Yaskawa INFORM job: OK_R2_O55B(90,0)KMOK_HARDOX.JBI

/JOB
//NAME OK_R2_O55B(90,0)KMOK_HARDOX
//POS
///NPOS 288,288,288,21,0,0
///TOOL 0
///POSTYPE PULSE
///PULSE
C00000=-9957,-80120,-66349,29251,62843,-41580
C00001=-119270,-98989,-86741,-6328,68520,-73858
C00002=-119780,-37820,-56111,-5839,80997,-74654
C00003=-120049,20077,-10457,-5740,82625,-74818
C00004=-144319,37014,-5855,2257,77898,-81650
C00005=-140529,51042,7974,-9565,85073,-64090
C00006=-140529,50609,8792,-9570,84355,-64035
C00007=-140529,50663,8686,-9570,84448,-64042
C00008=-140735,53191,11473,-9511,84012,-64075
C00009=-140529,50663,8686,-9570,84448,-64042
C00010=-132608,43274,6223,-26925,79302,-63189
C00011=-133562,42203,5091,-26579,79144,-63498
C00012=-132608,43724,5035,-26857,80165,-63389
C00013=-141550,80814,37938,-2920,95813,-64462
C00014=-141396,81120,39088,-2939,95269,-64399
C00015=-141396,80823,39851,-2936,94645,-64387
C00016=-141396,80877,39711,-2936,94757,-64389
C00017=-141226,78223,36470,-2964,95394,-64348
C00018=-141396,80877,39711,-2936,94757,-64389
C00019=-140829,81512,40491,-3016,94624,-64202
C00020=-140134,82102,41214,-3116,94504,-63971
C00021=-140829,81912,39485,-3022,95448,-64222
C00022=-137405,-31621,-64154,-15278,80257,-65243
C00023=-140140,-48602,-70983,-11254,71048,-74410
C00024=-141076,-49933,-70540,-10875,69988,-74633
C00025=-141076,-50277,-69406,-10930,69130,-74550
C00026=-141076,-50226,-69587,-10919,69267,-74563
C00027=-141467,-47373,-67920,-10702,69651,-74733
C00028=-141076,-50226,-69587,-10919,69267,-74563
C00029=-141874,-50689,-69854,-10542,69093,-74827
C00030=-143117,-51074,-70075,-9948,68881,-75243
C00031=-141874,-50354,-70946,-10488,69924,-74901
C00032=-147268,-6347,-50211,3630,100062,-76353
C00033=-146938,-6418,-49322,3551,99466,-76267
C00034=-146938,-6964,-48693,3545,98802,-76289
C00035=-146938,-6869,-48804,3545,98917,-76285
C00036=-146728,-9231,-50671,3485,98843,-76222
C00037=-146938,-6869,-48804,3545,98917,-76285
C00038=-151923,-27684,-59821,11781,84663,-77431
C00039=-150653,-27440,-59655,11346,84518,-77042
C00040=-151923,-26904,-61083,11768,85817,-77322
C00041=-127144,-21020,-54073,-16205,79799,-73423
C00042=-126838,-21905,-54390,-16337,79609,-73295
C00043=-126838,-22307,-53617,-16368,78953,-73207
C00044=-126838,-22196,-53838,-16359,79138,-73232
C00045=-124787,-22488,-54046,-17172,79509,-72603
C00046=-124787,-22654,-53716,-17186,79233,-72564
C00047=-125689,-22541,-53635,-16830,79066,-72840
C00048=-125495,-21030,-56345,-16804,81448,-73105
C00049=-137099,-135087,-110065,-14474,54639,-73776
C00050=-134884,-135911,-107803,-15875,53297,-72629
C00051=-134884,-134891,-106174,-15972,52835,-72554
C00052=-134884,-135228,-106712,-15940,52987,-72578
C00053=-129865,-136478,-107050,-18378,53628,-70507
C00054=-129865,-135962,-106251,-18430,53413,-70467
C00055=-131869,-135536,-106136,-17475,53114,-71287
C00056=-131377,-137376,-108864,-17542,53921,-71215
C00057=-139724,-149069,-111841,-14344,48265,-73992
C00058=-138735,-146286,-108991,-14933,48130,-73516
C00059=-138325,-143626,-108337,-14931,49139,-73488
C00060=-138410,-146030,-110862,-14819,49432,-73572
C00061=-176899,-100061,-98449,5916,63407,-89727
C00062=-179900,-97566,-95391,7380,63058,-90869
C00063=-179900,-97456,-94205,7424,62390,-90913
C00064=-179900,-97485,-94494,7413,62551,-90902
C00065=-169343,-119267,-96895,-8817,44711,-86747
C00066=-169343,-119018,-96376,-8846,44521,-86728
C00067=-168683,-117584,-95925,-9230,45055,-86464
C00068=-169216,-119583,-98076,-8807,45288,-86741
C00069=-162548,-60984,-74877,-11016,61707,-85538
C00070=-184352,-15408,-50569,-7993,71565,-76848
C00071=-184633,-15854,-49265,-7894,70519,-76872
C00072=-184633,-16240,-48510,-7925,69861,-76830
C00073=-184633,-16157,-48676,-7919,70004,-76840
C00074=-184233,-13625,-46764,-8123,70163,-76718
C00075=-184633,-16157,-48676,-7919,70004,-76840
C00076=-187381,11831,-34077,-2210,90888,-77611
C00077=-186375,11183,-34661,-2532,90938,-77309
C00078=-187381,12466,-34757,-2212,91632,-77624
C00079=-182192,42266,-7795,-19168,104635,-71349
C00080=-189067,53591,3425,-6745,109963,-71903
C00081=-189067,53103,3970,-6717,109382,-71871
C00082=-189067,53201,3857,-6722,109501,-71876
C00083=-189450,50860,1262,-6719,109865,-72023
C00084=-189067,53201,3857,-6722,109501,-71876
C00085=-185034,14321,-30270,-13993,89133,-70711
C00086=-186120,15304,-29370,-13637,88918,-71028
C00087=-185035,15000,-31072,-14012,89952,-70804
C00088=-182682,60735,12692,-23773,101105,-73169
C00089=-182682,60735,12692,-23773,101105,-73169
C00090=-183650,63040,17037,-21830,101290,-73190
C00091=-183650,62538,17836,-21764,100591,-73060
C00092=-183650,62598,17737,-21771,100675,-73076
C00093=-183528,62176,17250,-21794,100781,-73054
C00094=-183650,63460,16427,-21883,101838,-73293
C00095=-189227,48884,3,-21319,102940,-75405
C00096=-189468,47971,159,-21225,102357,-75379
C00097=-189468,47380,928,-21153,101633,-75249
C00098=-189468,47470,808,-21165,101744,-75269
C00099=-189367,47114,422,-21186,101818,-75248
C00100=-189432,48469,-714,-21310,103107,-75504
C00101=-175013,33301,-13153,-29999,98235,-49044
C00102=-175115,31766,-13036,-29901,97452,-48874
C00103=-175115,31283,-12339,-29848,96864,-48718
C00104=-175115,31366,-12461,-29858,96964,-48746
C00105=-176020,31704,-12122,-29658,96640,-48987
C00106=-175115,31366,-12461,-29858,96964,-48746
C00107=-177389,49548,3663,-27032,106629,-51330
C00108=-177525,47289,1207,-27077,106904,-51447
C00109=-177389,50188,2794,-27172,107402,-51519
C00110=-188015,41028,-12957,-12549,102183,-51760
C00111=-188146,40613,-11827,-12473,101279,-51708
C00112=-188165,40048,-11193,-12432,100612,-51645
C00113=-188165,40130,-11271,-12438,100700,-51655
C00114=-187344,39553,-11878,-12615,100887,-51416
C00115=-188165,40130,-11271,-12438,100700,-51655
C00116=-187875,42015,-9279,-12487,100489,-51542
C00117=-187566,44182,-6969,-12539,100230,-51416
C00118=-187875,42842,-10030,-12532,101356,-51631
C00119=-171459,-4614,-45398,-33605,84930,-48191
C00120=-170900,-6042,-43653,-33882,83616,-47589
C00121=-170900,-6530,-42846,-33920,82989,-47396
C00122=-170900,-6366,-43125,-33907,83204,-47461
C00123=-169534,-6797,-43470,-34394,83698,-47104
C00124=-169534,-7027,-43077,-34411,83398,-47011
C00125=-170096,-6658,-42784,-34212,83197,-47160
C00126=-169785,-6714,-43972,-34288,83898,-47260
C00127=-170398,9353,-32178,-34027,84507,-47673
C00128=-170215,8790,-30856,-34141,83656,-47346
C00129=-170215,8459,-30301,-34168,83233,-47218
C00130=-170215,8580,-30507,-34158,83391,-47266
C00131=-168835,8055,-30970,-34644,83914,-46912
C00132=-168835,7853,-30623,-34659,83653,-46831
C00133=-169290,8275,-30251,-34499,83472,-46947
C00134=-169213,8760,-31391,-34484,84292,-47173
C00135=-186069,25736,-27642,1526,92687,-58921
C00136=-186694,24000,-25961,1734,90774,-59129
C00137=-186694,23425,-25397,1733,90131,-59136
C00138=-186694,23662,-25633,1733,90398,-59133
C00139=-187283,19938,-29188,1932,90686,-59306
C00140=-187283,19583,-28837,1932,90288,-59311
C00141=-187018,21055,-27442,1842,90183,-59234
C00142=-187095,21607,-28285,1869,90987,-59245
C00143=-183298,20097,-29492,20792,92835,-75129
C00144=-182431,19002,-28896,20491,91770,-75035
C00145=-182431,18218,-28039,20473,90895,-75182
C00146=-182431,18445,-28295,20478,91152,-75138
C00147=-182795,15268,-31245,20599,91404,-75212
C00148=-182795,14938,-30873,20592,91029,-75276
C00149=-182620,16002,-29895,20535,90939,-75235
C00150=-182918,16284,-31560,20654,92104,-75132
C00151=-186265,48055,-1212,11796,87124,-79966
C00152=-186965,48573,-100,12039,86806,-80215
C00153=-186965,47910,713,12044,85983,-80295
C00154=-186965,47988,613,12044,86082,-80285
C00155=-186694,50137,2964,11952,85709,-80238
C00156=-186965,47988,613,12044,86082,-80285
C00157=-183974,61337,12156,5178,92575,-80151
C00158=-184645,62112,13036,5353,92472,-80362
C00159=-183974,61852,11573,5182,93194,-80123
C00160=-179887,91143,39097,3384,105716,-79096
C00161=-179840,89635,38790,3370,105129,-79098
C00162=-179840,89143,39323,3359,104550,-79112
C00163=-179840,89220,39235,3359,104642,-79110
C00164=-180024,86327,35591,3386,105404,-79148
C00165=-179840,89220,39235,3359,104642,-79110
C00166=-186520,62301,10800,17886,95759,-79423
C00167=-185837,61712,10122,17722,95736,-79206
C00168=-186520,62996,10143,17919,96484,-79317
C00169=-174567,29627,-16130,-6089,77714,-79974
C00170=-174267,31304,-12949,-6249,76643,-79825
C00171=-179026,33960,-10363,-4044,76139,-81308
C00172=-179026,33960,-10363,-4044,76139,-81308
C00173=-174024,52452,5562,-15282,87335,-82643
C00174=-181124,73254,24397,-458,98517,-83064
C00175=-182896,88636,42871,4243,102910,-77228
C00176=-180140,85434,39000,4081,103513,-76295
C00177=-180140,85434,39000,4081,103513,-76295
C00178=-184647,66871,19208,14888,96534,-76534
C00179=-174267,31304,-12949,-6249,76643,-79825
C00180=-174494,31610,-14990,-6114,78032,-79964
C00181=-175013,33301,-13153,-29999,98235,-49044
C00182=-175343,30235,-14768,-29874,97621,-48999
C00183=-171906,8512,-28233,-36021,84269,-45281
C00184=-172758,8115,-27337,-35775,83319,-45298
C00185=-172255,16606,-19687,-35958,83238,-45074
C00186=-171987,21177,-15407,-36061,83112,-44927
C00187=-171987,21177,-15407,-36061,83112,-44927
C00188=-180391,49402,2354,-18177,99354,-48334
C00189=-181669,75195,30349,-14733,108937,-58802
C00190=-184056,79778,35948,-11160,112261,-59402
C00191=-184907,70087,24268,-11430,114320,-59912
C00192=-184907,70087,24268,-11430,114320,-59912
C00193=-179652,49581,2539,-22463,107252,-59131
C00194=-172758,8115,-27337,-35775,83319,-45298
C00195=-172634,8341,-28512,-35775,84058,-45486
C00196=-153759,-18914,-52407,-41335,92413,-41016
C00197=-152540,-20147,-51692,-41605,92133,-40401
C00198=-152993,-17865,-48148,-41450,91166,-40203
C00199=-159302,-18488,-48629,-39831,88393,-41734
C00200=-159302,-18488,-48629,-39831,88393,-41734
C00201=-166414,13220,-30767,-32137,108347,-48872
C00202=-176872,12138,-36686,-11233,108343,-73701
C00203=-180381,23244,-27161,-3143,115050,-73458
C00204=-177105,21284,-28961,-3234,115264,-72371
C00205=-177105,21284,-28961,-3234,115264,-72371
C00206=-175157,7036,-41533,-6172,108047,-57119
C00207=-152993,-17864,-48148,-41450,91166,-40203
C00208=-153162,-17915,-50375,-41466,92114,-40650
C00209=-157956,-50140,-75109,2057,72313,-66630
C00210=-160224,-49369,-73518,3152,71800,-67393
C00211=-160503,-46712,-70493,3295,71314,-67502
C00212=-152523,-45623,-69844,-552,71345,-64837
C00213=-152523,-45623,-69844,-552,71345,-64837
C00214=-148927,-14811,-56631,-4403,95378,-64978
C00215=-148763,-1156,-47820,-3788,104699,-80082
C00216=-148630,8941,-39588,-6498,110680,-80853
C00217=-152650,7748,-40640,-6101,110438,-82132
C00218=-152650,7748,-40640,-6101,110438,-82132
C00219=-155137,-28863,-64381,-3266,86260,-82126
C00220=-160503,-46712,-70493,3295,71314,-67502
C00221=-160802,-46385,-74012,3397,73655,-67536
C00222=-183650,63040,17037,-21830,101290,-73190
C00223=-181574,69704,24792,-21980,100549,-72331
C00224=-183403,72450,28416,-19365,101992,-72790
C00225=-183309,72093,27990,-19380,102088,-72773
C00226=-183520,72890,28942,-19345,101875,-72811
C00227=-183958,70615,26232,-19347,102249,-73025
C00228=-183958,70934,25678,-19391,102726,-73103
C00229=-192384,50426,1269,-3472,96407,-72620
C00230=-192384,50016,1751,-3467,95901,-72606
C00231=-184117,69898,25781,-20658,102920,-73473
C00232=-190944,51922,5194,-20323,104561,-76131
C00233=-191415,50867,4029,-20288,104619,-76303
C00234=-193520,46467,-770,-20112,104798,-77054
C00235=-193520,47017,-1447,-20188,105457,-77168
C00236=-171741,3085,-44079,-22866,113958,-71236
C00237=-130348,29463,-19685,-22297,122832,-57661
C00238=-129735,-75595,-89571,-13565,72601,-49374
C00239=-143928,-62129,-81754,5565,77375,-52115
C00240=-142081,-63272,-82268,4854,76992,-51525
C00241=-142081,-63272,-82268,4854,76992,-51525
C00242=-127755,-87223,-86704,-10460,53798,-73673
C00243=-115599,-84167,-82164,-28839,54869,-69627
C00244=-115830,-77465,-79174,-28196,56209,-70126
C00245=-120569,18950,-14128,-20651,63759,-73413
C00246=-120570,21073,-12131,-20673,63629,-73389
C00247=-120570,21641,-13746,-20463,64836,-73615
C00248=-131610,1281,-36986,-13629,66366,-77786
C00249=-142543,23012,-23162,1458,80523,-80349
C00250=-139525,20137,-20065,-7610,74683,-81021
C00251=-142876,20525,-19823,1343,74165,-80532
C00252=-139662,22596,-17854,-198,73998,-79499
C00253=-139662,22596,-17854,-198,73998,-79499
C00254=-141793,37019,-7971,5655,84578,-79297
C00255=-137277,64767,17706,-3970,99490,-79285
C00256=-134924,69316,23645,-11495,101419,-79759
C00257=-137432,66658,20404,-11237,101707,-80615
C00258=-137432,66658,20404,-11237,101707,-80615
C00259=-140896,36331,-9506,-5892,87094,-79888
C00260=-139525,20137,-20065,-7610,74683,-81021
C00261=-139348,19632,-23053,-7644,76265,-81063
C00262=-132254,-67818,-87549,-11183,71854,-78389
C00263=-159615,-10281,-58898,-7636,100535,-90235
C00264=-166998,7770,-33829,-38669,93984,-50545
C00265=-168265,5123,-34621,-38271,92780,-50607
C00266=-168071,5758,-34073,-38323,92849,-50556
C00267=-167928,7434,-32586,-38359,92864,-50506
C00268=-172719,9530,-31332,-27823,83706,-47451
C00269=-172719,9530,-31332,-27823,83706,-47451
C00270=-172320,11286,-29764,-27974,83774,-47329
C00271=-179459,29271,-20356,-13837,95701,-48796
C00272=-183465,26284,-23592,-4892,94989,-48302
C00273=-181920,25197,-24652,-5328,95168,-47844
C00274=-174479,31677,-20338,1503,103987,-43795
C00275=-180212,26004,-22183,17305,100653,-42977
C00276=-181024,26764,-23793,17575,102127,-43022
C00277=-174949,-10425,-55605,-83,88665,-45823
C00278=-166426,-64689,-90076,-3246,82158,-43137
C00279=-131468,-82914,-92239,-33517,76500,-33632
C00280=-132751,-79712,-87299,-33282,74833,-33639
C00281=-135289,-78928,-86943,-32417,74029,-34418
C00282=-167985,-50339,-72512,-17957,69595,-45682
C00283=-161662,-56646,-68227,-34204,59627,-42917
C00284=-161369,-58109,-70614,-34130,60339,-43034
C00285=-153489,-114383,-104764,-40748,57378,-38072
C00286=-152369,-109512,-103102,-40646,59036,-38246
C00287=-7483,-109512,-100434,-40646,59036,-38246
BC00000=15,674025,1075175
BC00001=140466,674228,172767
BC00002=140466,729284,172767
BC00003=140466,791751,172767
BC00004=182866,791751,67340
BC00005=182866,791751,67340
BC00006=182866,791751,67340
BC00007=182866,791751,67340
BC00008=182866,791751,67340
BC00009=182866,791751,67340
BC00010=182866,791751,67340
BC00011=182866,791751,67340
BC00012=182866,791751,67340
BC00013=182866,791751,67340
BC00014=182866,791751,67340
BC00015=182866,791751,67340
BC00016=182866,791751,67340
BC00017=182866,791751,67340
BC00018=182866,791751,67340
BC00019=182866,791751,67340
BC00020=182866,791751,67340
BC00021=182866,791751,67340
BC00022=182866,791752,67339
BC00023=182866,791752,67339
BC00024=182866,791752,67339
BC00025=182866,791752,67339
BC00026=182866,791752,67339
BC00027=182866,791752,67339
BC00028=182866,791752,67339
BC00029=182866,791752,67339
BC00030=182866,791752,67339
BC00031=182866,791752,67339
BC00032=182866,791752,67339
BC00033=182866,791752,67339
BC00034=182866,791752,67339
BC00035=182866,791752,67339
BC00036=182866,791752,67337
BC00037=182866,791752,67339
BC00038=182866,791752,67339
BC00039=182866,791752,67339
BC00040=182866,791752,67339
BC00041=182866,791752,67339
BC00042=182866,791752,67339
BC00043=182866,791752,67339
BC00044=182866,791752,67339
BC00045=182866,791752,67339
BC00046=182866,791752,67339
BC00047=182866,791752,67339
BC00048=182866,791752,67339
BC00049=182866,791752,67339
BC00050=182866,791752,67339
BC00051=182866,791752,67339
BC00052=182866,791752,67339
BC00053=182866,791752,67339
BC00054=182866,791752,67339
BC00055=182866,791752,67339
BC00056=182866,791752,67339
BC00057=182866,791752,67339
BC00058=182866,791752,67339
BC00059=182866,791752,67339
BC00060=182866,791752,67339
BC00061=182866,791752,67339
BC00062=182866,791752,67339
BC00063=182866,791752,67339
BC00064=182866,791752,67339
BC00065=182866,791752,67339
BC00066=182866,791752,67339
BC00067=182865,791751,67336
BC00068=182865,791751,67336
BC00069=182865,791751,67336
BC00070=248959,799596,47476
BC00071=248959,799596,47476
BC00072=248959,799596,47476
BC00073=248959,799596,47476
BC00074=248959,799596,47476
BC00075=248959,799596,47476
BC00076=248959,799596,47476
BC00077=248959,799596,47476
BC00078=248959,799596,47476
BC00079=248959,799596,47476
BC00080=248959,799596,47476
BC00081=248959,799596,47476
BC00082=248959,799596,47476
BC00083=248959,799596,47476
BC00084=248959,799596,47476
BC00085=248959,799596,47476
BC00086=248959,799596,47476
BC00087=248959,799596,47475
BC00088=248959,799596,47475
BC00089=248959,799596,47475
BC00090=248959,799596,47475
BC00091=248959,799596,47475
BC00092=248959,799596,47475
BC00093=248959,799596,47475
BC00094=248959,799596,47475
BC00095=248959,799596,47475
BC00096=248959,799596,47475
BC00097=248959,799596,47475
BC00098=248959,799596,47475
BC00099=248959,799596,47475
BC00100=248959,799596,47475
BC00101=203274,799596,47475
BC00102=203274,799596,47475
BC00103=203274,799596,47475
BC00104=203274,799596,47475
BC00105=203274,799596,47475
BC00106=203274,799596,47475
BC00107=203274,799596,47475
BC00108=203274,799596,47475
BC00109=203274,799596,47475
BC00110=209362,813826,28785
BC00111=209362,813826,28785
BC00112=209362,813826,28785
BC00113=209362,813826,28785
BC00114=209362,813826,28785
BC00115=209362,813826,28785
BC00116=209362,813826,28785
BC00117=209362,813826,28784
BC00118=209362,813826,28785
BC00119=209362,813826,28785
BC00120=209362,813826,28785
BC00121=209362,813826,28785
BC00122=209362,813826,28785
BC00123=209362,813826,28785
BC00124=209362,813826,28785
BC00125=209362,813826,28785
BC00126=209362,813826,28785
BC00127=209362,813826,28785
BC00128=209362,813826,28785
BC00129=209362,813826,28785
BC00130=209362,813826,28785
BC00131=209362,813826,28785
BC00132=209362,813826,28785
BC00133=209362,813826,28785
BC00134=209362,813826,28785
BC00135=209362,813826,28784
BC00136=209362,813826,28784
BC00137=209362,813826,28784
BC00138=209362,813826,28784
BC00139=209362,813826,28784
BC00140=209362,813826,28784
BC00141=209362,813826,28784
BC00142=209362,813826,28784
BC00143=209362,813826,28784
BC00144=209362,813826,28784
BC00145=209362,813826,28784
BC00146=209362,813826,28784
BC00147=209362,813826,28784
BC00148=209362,813826,28784
BC00149=209362,813826,28784
BC00150=209362,813826,28784
BC00151=209363,813827,28780
BC00152=209363,813827,28780
BC00153=209363,813827,28780
BC00154=209363,813827,28780
BC00155=209363,813827,28780
BC00156=209363,813827,28780
BC00157=209363,813827,28780
BC00158=209363,813827,28780
BC00159=209363,813827,28780
BC00160=209363,813827,1884
BC00161=209363,813827,1884
BC00162=209363,813827,1884
BC00163=209363,813827,1884
BC00164=209363,813827,1884
BC00165=209363,813827,1884
BC00166=209363,813827,1884
BC00167=209363,813827,1884
BC00168=209363,813827,1884
BC00169=209363,813827,28780
BC00170=209363,813827,28780
BC00171=209363,813827,28780
BC00172=209363,813827,28780
BC00173=209363,813827,28780
BC00174=209363,813827,28780
BC00175=209363,813827,28776
BC00176=209363,813827,28776
BC00177=209363,813827,28776
BC00178=209363,813827,28776
BC00179=209363,813827,28780
BC00180=209363,813827,28780
BC00181=203274,799596,47475
BC00182=203274,799596,47475
BC00183=203274,799596,47475
BC00184=203274,799596,47475
BC00185=203274,799596,47475
BC00186=203275,799597,47472
BC00187=203275,799597,47472
BC00188=203275,799597,47472
BC00189=203275,799597,47471
BC00190=203275,799597,47471
BC00191=203275,799597,47470
BC00192=203275,799597,47470
BC00193=203275,799597,47470
BC00194=203274,799596,47475
BC00195=203275,799596,47475
BC00196=203275,799596,47475
BC00197=203275,799596,47474
BC00198=203275,799596,47474
BC00199=203275,799596,47474
BC00200=203275,799596,47474
BC00201=203275,799596,47474
BC00202=203275,799596,47474
BC00203=203275,799596,47474
BC00204=203275,799596,47474
BC00205=203275,799596,47474
BC00206=203275,799596,47474
BC00207=203275,799596,47474
BC00208=203275,799596,47474
BC00209=203275,799596,47474
BC00210=203275,799596,47474
BC00211=203275,799596,47474
BC00212=203275,799596,47474
BC00213=203275,799596,47474
BC00214=203275,799596,47474
BC00215=203275,799596,47474
BC00216=203275,799596,47474
BC00217=203275,799596,47474
BC00218=203275,799596,47474
BC00219=203275,799596,47474
BC00220=203275,799596,47474
BC00221=203275,799596,47474
BC00222=248959,799596,47475
BC00223=248959,799596,47475
BC00224=248959,799596,47475
BC00225=248959,799596,47475
BC00226=248959,799596,47475
BC00227=248959,799596,47475
BC00228=248959,799596,47475
BC00229=248959,799596,47475
BC00230=248959,799596,47475
BC00231=248959,799596,47475
BC00232=248959,799596,47475
BC00233=248959,799596,47475
BC00234=248959,799596,47475
BC00235=248959,799596,47475
BC00236=248959,799596,47475
BC00237=169428,732562,47475
BC00238=169431,732564,47474
BC00239=169431,732564,47474
BC00240=169431,732564,47474
BC00241=169431,732564,47474
BC00242=169431,732564,47474
BC00243=169431,732564,47474
BC00244=169431,732564,47474
BC00245=172916,732564,47474
BC00246=172916,732564,47474
BC00247=172916,732564,47474
BC00248=172916,804432,47474
BC00249=172916,804432,47474
BC00250=172916,804432,47473
BC00251=172916,804432,47473
BC00252=172916,804432,47473
BC00253=172916,804432,47473
BC00254=172916,804432,47473
BC00255=172916,804432,47473
BC00256=172916,804432,47473
BC00257=172916,804432,47473
BC00258=172916,804432,47473
BC00259=172916,804432,47473
BC00260=172916,804432,47473
BC00261=172916,804432,47473
BC00262=172916,804432,47473
BC00263=172916,804432,47473
BC00264=209362,813826,28785
BC00265=209362,813826,28785
BC00266=209362,813826,28785
BC00267=209362,813826,28785
BC00268=209362,813826,28785
BC00269=209362,813826,28785
BC00270=209362,813826,28785
BC00271=209362,813826,28785
BC00272=209362,813826,28785
BC00273=209362,813826,28785
BC00274=209362,813826,28785
BC00275=209362,813826,28785
BC00276=209362,813826,28785
BC00277=209362,813826,28785
BC00278=209362,813826,28785
BC00279=209362,755898,28785
BC00280=209362,755898,28785
BC00281=209362,755898,28785
BC00282=209362,755898,28785
BC00283=209362,755898,28785
BC00284=209362,755898,28785
BC00285=209362,755898,28785
BC00286=209362,675971,28785
BC00287=209362,663746,462190
EC00000=798156,0
EC00001=798153,2
EC00002=798153,2
EC00003=798153,2
EC00004=798153,2
EC00005=798153,2
EC00006=798153,2
EC00007=798153,2
EC00008=798153,2
EC00009=798153,2
EC00010=798153,2
EC00011=798153,2
EC00012=798153,2
EC00013=798153,2
EC00014=798153,2
EC00015=798153,2
EC00016=798153,2
EC00017=798153,2
EC00018=798153,2
EC00019=798153,2
EC00020=798153,2
EC00021=798153,2
EC00022=798152,3
EC00023=798152,3
EC00024=798152,3
EC00025=798152,3
EC00026=798152,3
EC00027=798152,3
EC00028=798152,3
EC00029=798152,3
EC00030=798152,3
EC00031=798152,3
EC00032=798152,3
EC00033=798152,3
EC00034=798152,3
EC00035=798152,3
EC00036=798151,3
EC00037=798152,3
EC00038=798152,3
EC00039=798152,3
EC00040=798152,3
EC00041=798152,3
EC00042=798152,3
EC00043=798152,3
EC00044=798152,3
EC00045=798152,3
EC00046=798152,3
EC00047=798152,3
EC00048=798152,3
EC00049=798152,3
EC00050=798152,3
EC00051=798152,3
EC00052=798152,3
EC00053=798152,3
EC00054=798152,3
EC00055=798152,3
EC00056=798152,3
EC00057=798152,3
EC00058=798152,3
EC00059=798152,3
EC00060=798152,3
EC00061=798152,3
EC00062=798152,3
EC00063=798152,3
EC00064=798152,3
EC00065=798152,3
EC00066=798152,3
EC00067=798151,3
EC00068=798151,3
EC00069=798151,3
EC00070=798151,3
EC00071=798151,3
EC00072=798151,3
EC00073=798151,3
EC00074=798151,3
EC00075=798151,3
EC00076=798151,3
EC00077=798151,3
EC00078=798151,3
EC00079=798151,3
EC00080=798151,3
EC00081=798151,3
EC00082=798151,3
EC00083=798151,3
EC00084=798151,3
EC00085=798151,3
EC00086=798151,3
EC00087=798150,4
EC00088=798150,4
EC00089=798150,4
EC00090=798150,4
EC00091=798150,4
EC00092=798150,4
EC00093=798150,4
EC00094=798150,4
EC00095=798150,4
EC00096=798150,4
EC00097=798149,4
EC00098=798149,4
EC00099=798149,4
EC00100=798149,4
EC00101=798148,4
EC00102=798148,4
EC00103=798148,4
EC00104=798148,4
EC00105=798148,4
EC00106=798148,4
EC00107=798148,4
EC00108=798148,4
EC00109=798148,4
EC00110=798148,4
EC00111=798148,4
EC00112=798148,4
EC00113=798148,4
EC00114=798148,4
EC00115=798148,4
EC00116=798148,4
EC00117=798147,5
EC00118=798148,4
EC00119=798148,4
EC00120=798148,4
EC00121=798148,4
EC00122=798148,4
EC00123=798148,4
EC00124=798148,4
EC00125=798148,4
EC00126=798148,4
EC00127=798148,4
EC00128=798148,4
EC00129=798148,4
EC00130=798148,4
EC00131=798148,4
EC00132=798148,4
EC00133=798148,4
EC00134=798148,4
EC00135=798147,4
EC00136=798147,4
EC00137=798147,4
EC00138=798147,4
EC00139=798147,4
EC00140=798147,4
EC00141=798147,4
EC00142=798147,4
EC00143=798147,4
EC00144=798147,4
EC00145=798147,4
EC00146=798147,4
EC00147=798147,4
EC00148=798147,4
EC00149=798147,4
EC00150=798147,4
EC00151=798145,8
EC00152=798145,8
EC00153=798145,8
EC00154=798145,8
EC00155=798145,8
EC00156=798145,8
EC00157=798145,8
EC00158=798145,8
EC00159=798145,8
EC00160=798145,8
EC00161=798145,8
EC00162=798145,8
EC00163=798145,8
EC00164=798145,8
EC00165=798145,8
EC00166=798145,8
EC00167=798145,8
EC00168=798145,8
EC00169=798145,8
EC00170=798145,8
EC00171=798145,11
EC00172=798145,11
EC00173=798145,11
EC00174=798145,11
EC00175=798144,11
EC00176=798144,11
EC00177=798144,11
EC00178=798144,11
EC00179=798145,8
EC00180=798145,8
EC00181=798148,4
EC00182=798148,4
EC00183=798148,4
EC00184=798148,4
EC00185=798148,4
EC00186=798147,4
EC00187=798147,4
EC00188=798147,4
EC00189=798145,5
EC00190=798145,5
EC00191=798144,6
EC00192=798144,6
EC00193=798144,6
EC00194=798148,4
EC00195=798147,4
EC00196=798147,4
EC00197=798146,5
EC00198=798146,5
EC00199=798146,5
EC00200=798146,5
EC00201=798146,5
EC00202=798146,5
EC00203=798146,5
EC00204=798146,5
EC00205=798146,5
EC00206=798146,5
EC00207=798146,5
EC00208=798146,5
EC00209=798146,5
EC00210=798146,5
EC00211=798146,5
EC00212=798146,5
EC00213=798146,5
EC00214=798146,5
EC00215=798146,5
EC00216=798146,5
EC00217=798146,5
EC00218=798146,5
EC00219=798146,5
EC00220=798146,5
EC00221=798146,5
EC00222=798150,4
EC00223=798150,4
EC00224=798150,4
EC00225=798150,4
EC00226=798150,4
EC00227=798150,4
EC00228=798150,4
EC00229=798150,4
EC00230=798150,4
EC00231=798150,4
EC00232=798150,4
EC00233=798150,4
EC00234=798150,4
EC00235=798150,4
EC00236=798150,4
EC00237=798150,4
EC00238=798148,13
EC00239=798148,13
EC00240=798148,13
EC00241=798148,13
EC00242=798148,13
EC00243=798148,13
EC00244=798148,13
EC00245=798148,13
EC00246=798148,13
EC00247=798148,13
EC00248=798148,13
EC00249=798148,13
EC00250=798147,13
EC00251=798147,13
EC00252=798147,13
EC00253=798147,13
EC00254=798147,13
EC00255=798147,13
EC00256=798147,13
EC00257=798147,13
EC00258=798147,13
EC00259=798147,13
EC00260=798147,13
EC00261=798147,13
EC00262=798147,13
EC00263=798147,13
EC00264=798148,4
EC00265=798148,4
EC00266=798148,4
EC00267=798148,4
EC00268=798148,4
EC00269=798148,4
EC00270=798148,4
EC00271=798148,4
EC00272=798148,4
EC00273=798148,4
EC00274=798148,4
EC00275=798148,4
EC00276=798148,4
EC00277=798148,4
EC00278=798148,4
EC00279=798148,4
EC00280=798148,4
EC00281=798148,4
EC00282=798148,4
EC00283=798148,4
EC00284=798148,4
EC00285=798148,4
EC00286=798148,4
EC00287=798148,4
///POSTYPE BASE
///RECTAN
///RCONF 0,0,0,0,0,0,0,0,0,0,0,0,0,0,0,0,0,0,0,0,0,0,0,0
P00006=0.222,-3.123,-1.508,0.0000,0.0000,0.0000
P00021=-0.225,-6.128,-0.405,0.0000,0.0000,0.0000
P00022=0.222,-3.123,-1.508,0.0000,0.0000,0.0000
P00023=0.143,-0.036,0.682,0.0000,0.0000,0.0000
P00024=0.145,-0.552,1.326,0.0000,0.0000,0.0000
P00025=-2.003,0.006,0.728,0.0000,0.0000,0.0000
P00026=0.562,-0.002,-0.337,0.0000,0.0000,0.0000
P00027=-0.746,0.015,-9.096,0.0000,0.0000,0.0000
P00028=-2.237,-0.018,-7.702,0.0000,0.0000,0.0000
P00029=-2.156,-0.086,-4.681,0.0000,0.0000,0.0000
P00030=5.926,-4.294,-1.390,0.0000,0.0000,0.0000
P00031=1.853,-0.001,-1.549,0.0000,0.0000,0.0000
P00032=1.957,0.503,-7.217,0.0000,0.0000,0.0000
///RCONF 0,0,0,0,1,0,0,0,0,0,0,0,0,0,0,0,0,0,0,0,0,0,0,0
P00033=-0.123,0.612,-5.012,0.0000,0.0000,0.0000
///RCONF 0,0,0,0,0,0,0,0,0,0,0,0,0,0,0,0,0,0,0,0,0,0,0,0
P00034=-0.304,0.773,-2.693,0.0000,0.0000,0.0000
P00035=2.817,0.591,-1.622,0.0000,0.0000,0.0000
P00036=-1.108,-0.829,1.850,0.0000,0.0000,0.0000
P00037=0.023,0.937,-2.677,0.0000,0.0000,0.0000
P00038=0.158,-1.133,-1.952,0.0000,0.0000,0.0000
P00039=0.012,-3.081,-0.106,0.0000,0.0000,0.0000
P00040=-0.030,9.648,2.467,0.0000,0.0000,0.0000
//INST
///DATE 2025/01/24 15:35
///ATTR SC,RW
///GROUP1 RB1,BS1
///GROUP2 ST1
NOP
'MUZYLO 310124
'POPRAWA I SPAWANIE
'OK_R2_o55b(90,0)
'
'Path S3809
SFTOF3D
MOVJ C00000 BC00000 VJ=100.00  +MOVJ EC00000 VJ=100.00
CALL JOB:CLEAN-R1_KM_3P
MOVJ C00001 BC00001 VJ=100.00  +MOVJ EC00001 VJ=100.00
MOVL C00002 BC00002 V=666.7  +MOVJ EC00002 VJ=100.00
MOVL C00003 BC00003 V=666.7  +MOVJ EC00003 VJ=100.00
MOVL C00004 BC00004 V=666.7  +MOVJ EC00004 VJ=100.00
SMOVL C00005 BC00005 V=166.7  +MOVJ EC00005
SREFP 3 C00006 BC00006  +REFP EC00006
CALL JOB:SEARCH-R1-S13D
SET P021 P006
SFTON3D P021
SMOVL C00007 BC00007 V=166.7  +MOVJ EC00007
SREFP 3 C00008 BC00008  +REFP EC00008
CALL JOB:SEARCH-R1-S13D
SET P021 P006
SFTON3D P021
SMOVL C00009 BC00009 V=166.7  +MOVJ EC00009
SMOVL C00010 BC00010 V=166.7  +MOVJ EC00010
SREFP 3 C00011 BC00011  +REFP EC00011
CALL JOB:SEARCH-R1-S13D
SET P021 P006
SFTON3D P021
SMOVL C00012 BC00012 V=166.7  +MOVJ EC00012
MOVL C00013 BC00013 V=666.7  +MOVJ EC00013 VJ=100.00
SMOVL C00014 BC00014 V=166.7  +MOVJ EC00014
SREFP 3 C00015 BC00015  +REFP EC00015
CALL JOB:SEARCH-R1-S13D
SET P022 P006
SFTON3D P022
SMOVL C00016 BC00016 V=166.7  +MOVJ EC00016
SREFP 3 C00017 BC00017  +REFP EC00017
CALL JOB:SEARCH-R1-S13D
SET P022 P006
SFTON3D P022
SMOVL C00018 BC00018 V=166.7  +MOVJ EC00018
SMOVL C00019 BC00019 V=166.7  +MOVJ EC00019
SREFP 3 C00020 BC00020  +REFP EC00020
CALL JOB:SEARCH-R1-S13D
SET P022 P006
SFTON3D P022
SMOVL C00021 BC00021 V=166.7  +MOVJ EC00021
SFTOF3D
MOVL C00022 BC00022 V=666.7  +MOVJ EC00022 VJ=100.00
MOVL C00023 BC00023 V=666.7  +MOVJ EC00023 VJ=100.00
SMOVL C00024 BC00024 V=166.7  +MOVJ EC00024
SREFP 3 C00025 BC00025  +REFP EC00025
CALL JOB:SEARCH-R1-S13D
SET P023 P006
SFTON3D P023
SMOVL C00026 BC00026 V=166.7  +MOVJ EC00026
SREFP 3 C00027 BC00027  +REFP EC00027
CALL JOB:SEARCH-R1-S13D
SET P023 P006
SFTON3D P023
SMOVL C00028 BC00028 V=166.7  +MOVJ EC00028
SMOVL C00029 BC00029 V=166.7  +MOVJ EC00029
SREFP 3 C00030 BC00030  +REFP EC00030
CALL JOB:SEARCH-R1-S13D
SET P023 P006
SFTON3D P023
SMOVL C00031 BC00031 V=166.7  +MOVJ EC00031
MOVL C00032 BC00032 V=666.7  +MOVJ EC00032 VJ=100.00
SMOVL C00033 BC00033 V=166.7  +MOVJ EC00033
SREFP 3 C00034 BC00034  +REFP EC00034
CALL JOB:SEARCH-R1-S13D
SET P024 P006
SFTON3D P024
SMOVL C00035 BC00035 V=166.7  +MOVJ EC00035
SREFP 3 C00036 BC00036  +REFP EC00036
CALL JOB:SEARCH-R1-S13D
SET P024 P006
SFTON3D P024
SMOVL C00037 BC00037 V=166.7  +MOVJ EC00037
SMOVL C00038 BC00038 V=166.7  +MOVJ EC00038
SREFP 3 C00039 BC00039  +REFP EC00039
CALL JOB:SEARCH-R1-S13D
SET P024 P006
SFTON3D P024
SMOVL C00040 BC00040 V=166.7  +MOVJ EC00040
SFTOF3D
MOVL C00041 BC00041 V=666.7  +MOVJ EC00041 VJ=100.00
SMOVL C00042 BC00042 V=166.7  +MOVJ EC00042
SREFP 3 C00043 BC00043  +REFP EC00043
CALL JOB:SEARCH-R1-S13D
SET P025 P006
SFTON3D P025
SMOVL C00044 BC00044 V=166.7  +MOVJ EC00044
SMOVL C00045 BC00045 V=166.7  +MOVJ EC00045
SMOVL C00046 BC00046 V=166.7  +MOVJ EC00046
SREFP 3 C00047 BC00047  +REFP EC00047
CALL JOB:SEARCH-R1-S13D
SET P025 P006
SFTON3D P025
SMOVL C00048 BC00048 V=166.7  +MOVJ EC00048
SFTOF3D
MOVL C00049 BC00049 V=666.7  +MOVJ EC00049 VJ=100.00
SMOVL C00050 BC00050 V=166.7  +MOVJ EC00050
SREFP 3 C00051 BC00051  +REFP EC00051
CALL JOB:SEARCH-R1-S13D
SET P026 P006
SFTON3D P026
SMOVL C00052 BC00052 V=166.7  +MOVJ EC00052
SMOVL C00053 BC00053 V=166.7  +MOVJ EC00053
SMOVL C00054 BC00054 V=166.7  +MOVJ EC00054
SREFP 3 C00055 BC00055  +REFP EC00055
CALL JOB:SEARCH-R1-S13D
SET P026 P006
SFTON3D P026
SMOVL C00056 BC00056 V=166.7  +MOVJ EC00056
SMOVL C00057 BC00057 V=166.7  +MOVJ EC00057
SMOVL C00058 BC00058 V=166.7  +MOVJ EC00058
SREFP 3 C00059 BC00059  +REFP EC00059
CALL JOB:SEARCH-R1-S13D
SET P027 P006
SFTON3D P027
SMOVL C00060 BC00060 V=166.7  +MOVJ EC00060
SFTOF3D
MOVL C00061 BC00061 V=666.7  +MOVJ EC00061 VJ=100.00
SMOVL C00062 BC00062 V=166.7  +MOVJ EC00062
SREFP 3 C00063 BC00063  +REFP EC00063
CALL JOB:SEARCH-R1-S13D
SET P028 P006
SFTON3D P028
SMOVL C00064 BC00064 V=166.7  +MOVJ EC00064
SMOVL C00065 BC00065 V=166.7  +MOVJ EC00065
SMOVL C00066 BC00066 V=166.7  +MOVJ EC00066
SREFP 3 C00067 BC00067  +REFP EC00067
CALL JOB:SEARCH-R1-S13D
SET P028 P006
SFTON3D P028
SMOVL C00068 BC00068 V=166.7  +MOVJ EC00068
SFTOF3D
SMOVL C00069 BC00069 V=666.7  +MOVJ EC00069
MOVL C00070 BC00070 V=666.7  +MOVJ EC00070 VJ=100.00
SMOVL C00071 BC00071 V=166.7  +MOVJ EC00071
SREFP 3 C00072 BC00072  +REFP EC00072
CALL JOB:SEARCH-R1-S13D
SET P029 P006
SFTON3D P029
SMOVL C00073 BC00073 V=166.7  +MOVJ EC00073
SREFP 3 C00074 BC00074  +REFP EC00074
CALL JOB:SEARCH-R1-S13D
SET P029 P006
SFTON3D P029
SMOVL C00075 BC00075 V=166.7  +MOVJ EC00075
SMOVL C00076 BC00076 V=166.7  +MOVJ EC00076
SREFP 3 C00077 BC00077  +REFP EC00077
CALL JOB:SEARCH-R1-S13D
SET P029 P006
SFTON3D P029
SMOVL C00078 BC00078 V=166.7  +MOVJ EC00078
MOVL C00079 BC00079 V=666.7  +MOVJ EC00079 VJ=100.00
SMOVL C00080 BC00080 V=166.7  +MOVJ EC00080
SREFP 3 C00081 BC00081  +REFP EC00081
CALL JOB:SEARCH-R1-S13D
SET P030 P006
SFTON3D P030
SMOVL C00082 BC00082 V=166.7  +MOVJ EC00082
SREFP 3 C00083 BC00083  +REFP EC00083
CALL JOB:SEARCH-R1-S13D
SET P030 P006
SFTON3D P030
SMOVL C00084 BC00084 V=166.7  +MOVJ EC00084
SMOVL C00085 BC00085 V=166.7  +MOVJ EC00085
SREFP 3 C00086 BC00086  +REFP EC00086
CALL JOB:SEARCH-R1-S13D
SET P030 P006
SFTON3D P030
SMOVL C00087 BC00087 V=166.7  +MOVJ EC00087
SMOVL C00088 BC00088 V=666.7  +MOVJ EC00088
SMOVL C00089 BC00089 V=666.7  +MOVJ EC00089
SMOVL C00090 BC00090 V=166.7  +MOVJ EC00090
SREFP 3 C00091 BC00091  +REFP EC00091
CALL JOB:SEARCH-R1-S13D
SET P031 P006
SFTON3D P031
SMOVL C00092 BC00092 V=166.7  +MOVJ EC00092
SREFP 3 C00093 BC00093  +REFP EC00093
CALL JOB:SEARCH-R1-S13D
SET P031 P006
SFTON3D P031
SMOVL C00094 BC00094 V=166.7  +MOVJ EC00094
SMOVL C00095 BC00095 V=666.7  +MOVJ EC00095
SMOVL C00096 BC00096 V=166.7  +MOVJ EC00096
SREFP 3 C00097 BC00097  +REFP EC00097
CALL JOB:SEARCH-R1-S13D
SET P032 P006
SFTON3D P032
SMOVL C00098 BC00098 V=166.7  +MOVJ EC00098
SREFP 3 C00099 BC00099  +REFP EC00099
CALL JOB:SEARCH-R1-S13D
SET P032 P006
SFTON3D P032
SMOVL C00100 BC00100 V=166.7  +MOVJ EC00100
SFTOF3D
MOVL C00101 BC00101 V=666.7  +MOVJ EC00101 VJ=100.00
SMOVL C00102 BC00102 V=166.7  +MOVJ EC00102
SREFP 3 C00103 BC00103  +REFP EC00103
CALL JOB:SEARCH-R1-S13D
SET P033 P006
SFTON3D P033
SMOVL C00104 BC00104 V=166.7  +MOVJ EC00104
SREFP 3 C00105 BC00105  +REFP EC00105
CALL JOB:SEARCH-R1-S13D
SET P033 P006
SFTON3D P033
SMOVL C00106 BC00106 V=166.7  +MOVJ EC00106
SMOVL C00107 BC00107 V=166.7  +MOVJ EC00107
SREFP 3 C00108 BC00108  +REFP EC00108
CALL JOB:SEARCH-R1-S13D
SET P033 P006
SFTON3D P033
SMOVL C00109 BC00109 V=166.7  +MOVJ EC00109
MOVL C00110 BC00110 V=666.7  +MOVJ EC00110 VJ=100.00
SMOVL C00111 BC00111 V=166.7  +MOVJ EC00111
SREFP 3 C00112 BC00112  +REFP EC00112
CALL JOB:SEARCH-R1-S13D
SET P034 P006
SFTON3D P034
SMOVL C00113 BC00113 V=166.7  +MOVJ EC00113
SREFP 3 C00114 BC00114  +REFP EC00114
CALL JOB:SEARCH-R1-S13D
SET P034 P006
SFTON3D P034
SMOVL C00115 BC00115 V=166.7  +MOVJ EC00115
SMOVL C00116 BC00116 V=166.7  +MOVJ EC00116
SREFP 3 C00117 BC00117  +REFP EC00117
CALL JOB:SEARCH-R1-S13D
SET P034 P006
SFTON3D P034
SMOVL C00118 BC00118 V=166.7  +MOVJ EC00118
MOVL C00119 BC00119 V=666.7  +MOVJ EC00119 VJ=0.78
SMOVL C00120 BC00120 V=166.7  +MOVJ EC00120
SREFP 3 C00121 BC00121  +REFP EC00121
CALL JOB:SEARCH-R1-S13D
SET P035 P006
SFTON3D P035
SMOVL C00122 BC00122 V=166.7  +MOVJ EC00122
SMOVL C00123 BC00123 V=166.7  +MOVJ EC00123
SMOVL C00124 BC00124 V=166.7  +MOVJ EC00124
SREFP 3 C00125 BC00125  +REFP EC00125
CALL JOB:SEARCH-R1-S13D
SET P035 P006
SFTON3D P035
SMOVL C00126 BC00126 V=166.7  +MOVJ EC00126
SMOVL C00127 BC00127 V=666.7  +MOVJ EC00127
SMOVL C00128 BC00128 V=166.7  +MOVJ EC00128
SREFP 3 C00129 BC00129  +REFP EC00129
CALL JOB:SEARCH-R1-S13D
SET P036 P006
SFTON3D P036
SMOVL C00130 BC00130 V=166.7  +MOVJ EC00130
SMOVL C00131 BC00131 V=166.7  +MOVJ EC00131
SMOVL C00132 BC00132 V=166.7  +MOVJ EC00132
SREFP 3 C00133 BC00133  +REFP EC00133
CALL JOB:SEARCH-R1-S13D
SET P036 P006
SFTON3D P036
SMOVL C00134 BC00134 V=166.7  +MOVJ EC00134
SMOVL C00135 BC00135 V=666.7  +MOVJ EC00135
SMOVL C00136 BC00136 V=166.7  +MOVJ EC00136
SREFP 3 C00137 BC00137  +REFP EC00137
CALL JOB:SEARCH-R1-S13D
SET P037 P006
SFTON3D P037
SMOVL C00138 BC00138 V=166.7  +MOVJ EC00138
SMOVL C00139 BC00139 V=166.7  +MOVJ EC00139
SMOVL C00140 BC00140 V=166.7  +MOVJ EC00140
SREFP 3 C00141 BC00141  +REFP EC00141
CALL JOB:SEARCH-R1-S13D
SET P037 P006
SFTON3D P037
SMOVL C00142 BC00142 V=166.7  +MOVJ EC00142
SMOVL C00143 BC00143 V=666.7  +MOVJ EC00143
SMOVL C00144 BC00144 V=166.7  +MOVJ EC00144
SREFP 3 C00145 BC00145  +REFP EC00145
CALL JOB:SEARCH-R1-S13D
SET P038 P006
SFTON3D P038
SMOVL C00146 BC00146 V=166.7  +MOVJ EC00146
SMOVL C00147 BC00147 V=166.7  +MOVJ EC00147
SMOVL C00148 BC00148 V=166.7  +MOVJ EC00148
SREFP 3 C00149 BC00149  +REFP EC00149
CALL JOB:SEARCH-R1-S13D
SET P038 P006
SFTON3D P038
SMOVL C00150 BC00150 V=166.7  +MOVJ EC00150
SMOVL C00151 BC00151 V=666.7  +MOVJ EC00151
SMOVL C00152 BC00152 V=166.7  +MOVJ EC00152
SREFP 3 C00153 BC00153  +REFP EC00153
CALL JOB:SEARCH-R1-S13D
SET P039 P006
SFTON3D P039
SMOVL C00154 BC00154 V=166.7  +MOVJ EC00154
SREFP 3 C00155 BC00155  +REFP EC00155
CALL JOB:SEARCH-R1-S13D
SET P039 P006
SFTON3D P039
SMOVL C00156 BC00156 V=166.7  +MOVJ EC00156
SMOVL C00157 BC00157 V=166.7  +MOVJ EC00157
SREFP 3 C00158 BC00158  +REFP EC00158
CALL JOB:SEARCH-R1-S13D
SET P039 P006
SFTON3D P039
SMOVL C00159 BC00159 V=166.7  +MOVJ EC00159
MOVL C00160 BC00160 V=666.7  +MOVJ EC00160 VJ=100.00
SMOVL C00161 BC00161 V=166.7  +MOVJ EC00161
SREFP 3 C00162 BC00162  +REFP EC00162
CALL JOB:SEARCH-R1-S13D
SET P040 P006
SFTON3D P040
SMOVL C00163 BC00163 V=166.7  +MOVJ EC00163
SREFP 3 C00164 BC00164  +REFP EC00164
CALL JOB:SEARCH-R1-S13D
SET P040 P006
SFTON3D P040
SMOVL C00165 BC00165 V=166.7  +MOVJ EC00165
SMOVL C00166 BC00166 V=166.7  +MOVJ EC00166
SREFP 3 C00167 BC00167  +REFP EC00167
CALL JOB:SEARCH-R1-S13D
SET P040 P006
SFTON3D P040
SMOVL C00168 BC00168 V=166.7  +MOVJ EC00168
SMOVL C00169 BC00169 V=666.7  +MOVJ EC00169
MACRO1 MJ#(0) ARGF9
SMOVL C00170 BC00170 V=166.7 PL=0  +MOVJ EC00170
ARCON
SFTON3D P039
SMOVL C00171 BC00171 V=11.7  +MOVJ EC00171
SMOVC C00172 BC00172 V=15.0  +MOVJ EC00172
SMOVC C00173 BC00173 V=15.0  +MOVJ EC00173
SMOVC C00174 BC00174 V=15.0  +MOVJ EC00174
SFTON3D P040
SMOVL C00175 BC00175 V=11.7  +MOVJ EC00175
SMOVL C00176 BC00176 V=11.7  +MOVJ EC00176
SMOVC C00177 BC00177 V=15.0  +MOVJ EC00177
SMOVC C00178 BC00178 V=15.0  +MOVJ EC00178
SMOVC C00179 BC00179 V=15.0  +MOVJ EC00179
ARCOF
SMOVL C00180 BC00180 V=166.7  +MOVJ EC00180
SFTOF3D
MOVL C00181 BC00181 V=666.7  +MOVJ EC00181 VJ=100.00
SMOVL C00182 BC00182 V=166.7  +MOVJ EC00182
SMOVL C00183 BC00183 V=166.7  +MOVJ EC00183
SFTON3D P033
SMOVL C00184 BC00184 V=166.7 PL=0  +MOVJ EC00184
ARCON
SFTON3D P034
SMOVL C00185 BC00185 V=11.7  +MOVJ EC00185
SMOVL C00186 BC00186 V=11.7  +MOVJ EC00186
SMOVC C00187 BC00187 V=15.0  +MOVJ EC00187
SMOVC C00188 BC00188 V=15.0  +MOVJ EC00188
SMOVC C00189 BC00189 V=15.0  +MOVJ EC00189
SFTON3D P033
SMOVL C00190 BC00190 V=11.7  +MOVJ EC00190
SMOVL C00191 BC00191 V=11.7  +MOVJ EC00191
SMOVC C00192 BC00192 V=15.0  +MOVJ EC00192
SMOVC C00193 BC00193 V=15.0  +MOVJ EC00193
SMOVC C00194 BC00194 V=15.0  +MOVJ EC00194
ARCOF
SMOVL C00195 BC00195 V=166.7  +MOVJ EC00195
SFTOF3D
SMOVL C00196 BC00196 V=666.7  +MOVJ EC00196
SFTON3D P029
SMOVL C00197 BC00197 V=166.7  +MOVJ EC00197
SMOVL C00198 BC00198 V=166.7 PL=0  +MOVJ EC00198
ARCON
SFTON3D P030
SMOVL C00199 BC00199 V=11.7  +MOVJ EC00199
SMOVC C00200 BC00200 V=15.0  +MOVJ EC00200
SMOVC C00201 BC00201 V=15.0  +MOVJ EC00201
SMOVC C00202 BC00202 V=15.0  +MOVJ EC00202
SFTON3D P029
SMOVL C00203 BC00203 V=11.7  +MOVJ EC00203
SMOVL C00204 BC00204 V=11.7  +MOVJ EC00204
SMOVC C00205 BC00205 V=15.0  +MOVJ EC00205
SMOVC C00206 BC00206 V=15.0  +MOVJ EC00206
SMOVC C00207 BC00207 V=15.0  +MOVJ EC00207
ARCOF
SMOVL C00208 BC00208 V=166.7  +MOVJ EC00208
SFTOF3D
SMOVL C00209 BC00209 V=666.7  +MOVJ EC00209
SMOVL C00210 BC00210 V=666.7  +MOVJ EC00210
SFTON3D P023
SMOVL C00211 BC00211 V=166.7 PL=0  +MOVJ EC00211
ARCON
SFTON3D P024
SMOVL C00212 BC00212 V=11.7  +MOVJ EC00212
SMOVC C00213 BC00213 V=15.0  +MOVJ EC00213
SMOVC C00214 BC00214 V=15.0  +MOVJ EC00214
SMOVC C00215 BC00215 V=15.0  +MOVJ EC00215
SFTON3D P023
SMOVL C00216 BC00216 V=11.7  +MOVJ EC00216
SMOVL C00217 BC00217 V=11.7  +MOVJ EC00217
SMOVC C00218 BC00218 V=15.0  +MOVJ EC00218
SMOVC C00219 BC00219 V=15.0  +MOVJ EC00219
SMOVC C00220 BC00220 V=15.0  +MOVJ EC00220
ARCOF
SMOVL C00221 BC00221 V=166.7  +MOVJ EC00221
PAUSE
SFTOF3D
SMOVL C00222 BC00222 V=666.7  +MOVJ EC00222
SFTON3D P031
SMOVL C00223 BC00223 V=666.7  +MOVJ EC00223
SMOVL C00224 BC00224 V=166.7 PL=0  +MOVJ EC00224
SREFP 1 C00225 BC00225  +REFP EC00225
SREFP 2 C00226 BC00226  +REFP EC00226
ARCON
SWVON WEV#(71)
SMOVL C00227 BC00227 V=6.7  +MOVJ EC00227
ARCOF
SWVOF
SMOVL C00228 BC00228 V=166.7  +MOVJ EC00228
SMOVL C00229 BC00229 V=166.7  +MOVJ EC00229
SMOVL C00230 BC00230 V=166.7 PL=0  +MOVJ EC00230
ARCON
SWVON WEV#(70)
SMOVL C00231 BC00231 V=6.7  +MOVJ EC00231
SFTON3D P032
SMOVL C00232 BC00232 V=6.7  +MOVJ EC00232
ARCOF
SWVOF
SMOVL C00233 BC00233 V=33.3 PL=0  +MOVJ EC00233
ARCON
SWVON WEV#(70)
SMOVL C00234 BC00234 V=6.7  +MOVJ EC00234
ARCOF
SWVOF
SMOVL C00235 BC00235 V=166.7  +MOVJ EC00235
SFTOF3D
SMOVL C00236 BC00236 V=666.7  +MOVJ EC00236
SMOVL C00237 BC00237 V=666.7  +MOVJ EC00237
SMOVL C00238 BC00238 V=666.7  +MOVJ EC00238
SFTON3D P027
SMOVL C00239 BC00239 V=166.7 PL=0  +MOVJ EC00239
ARCON
SMOVL C00240 BC00240 V=11.7  +MOVJ EC00240
SMOVC C00241 BC00241 V=15.0  +MOVJ EC00241
SMOVC C00242 BC00242 V=15.0  +MOVJ EC00242
SFTON3D P026
SMOVC C00243 BC00243 V=15.0  +MOVJ EC00243
SMOVL C00244 BC00244 V=11.7  +MOVJ EC00244
SFTON3D P025
SMOVL C00245 BC00245 V=11.7  +MOVJ EC00245
SMOVL C00246 BC00246 V=11.7  +MOVJ EC00246
ARCOF
SMOVL C00247 BC00247 V=166.7  +MOVJ EC00247
SFTOF3D
SMOVL C00248 BC00248 V=666.7  +MOVJ EC00248
SMOVL C00249 BC00249 V=666.7  +MOVJ EC00249
SFTON3D P021
SMOVL C00250 BC00250 V=166.7 PL=0  +MOVJ EC00250
ARCON
SFTON3D P022
SMOVL C00251 BC00251 V=11.7  +MOVJ EC00251
SMOVL C00252 BC00252 V=11.7  +MOVJ EC00252
SMOVC C00253 BC00253 V=15.0  +MOVJ EC00253
SMOVC C00254 BC00254 V=15.0  +MOVJ EC00254
SMOVC C00255 BC00255 V=15.0  +MOVJ EC00255
SFTON3D P021
SMOVL C00256 BC00256 V=11.7  +MOVJ EC00256
SMOVL C00257 BC00257 V=11.7  +MOVJ EC00257
SMOVC C00258 BC00258 V=15.0  +MOVJ EC00258
SMOVC C00259 BC00259 V=15.0  +MOVJ EC00259
SMOVC C00260 BC00260 V=15.0  +MOVJ EC00260
ARCOF
SMOVL C00261 BC00261 V=166.7  +MOVJ EC00261
SFTOF3D
MOVL C00262 BC00262 V=666.7  +MOVJ EC00262 VJ=0.78
MOVL C00263 BC00263 V=666.7  +MOVJ EC00263 VJ=0.78
SMOVL C00264 BC00264 V=666.7  +MOVJ EC00264
SFTON3D P035
SMOVL C00265 BC00265 V=166.7 PL=0  +MOVJ EC00265
ARCON
SMOVL C00266 BC00266 V=11.7  +MOVJ EC00266
SMOVL C00267 BC00267 V=11.7  +MOVJ EC00267
SFTON3D P036
SMOVL C00268 BC00268 V=11.7  +MOVJ EC00268
SMOVC C00269 BC00269 V=15.0  +MOVJ EC00269
SMOVC C00270 BC00270 V=15.0  +MOVJ EC00270
SFTON3D P037
SMOVC C00271 BC00271 V=15.0  +MOVJ EC00271
SMOVL C00272 BC00272 V=11.7  +MOVJ EC00272
SMOVL C00273 BC00273 V=11.7  +MOVJ EC00273
SFTON3D P038
SMOVL C00274 BC00274 V=11.7  +MOVJ EC00274
SMOVL C00275 BC00275 V=13.3  +MOVJ EC00275
ARCOF
SMOVL C00276 BC00276 V=166.7  +MOVJ EC00276
SFTOF3D
SMOVL C00277 BC00277 V=666.7  +MOVJ EC00277
SMOVL C00278 BC00278 V=666.7  +MOVJ EC00278
SMOVL C00279 BC00279 V=666.7  +MOVJ EC00279
SFTON3D P027
SMOVL C00280 BC00280 V=166.7 PL=0  +MOVJ EC00280
ARCON
SMOVL C00281 BC00281 V=11.7  +MOVJ EC00281
SFTON3D P028
SMOVL C00282 BC00282 V=11.7  +MOVJ EC00282
SMOVL C00283 BC00283 V=11.7  +MOVJ EC00283
ARCOF
SMOVL C00284 BC00284 V=166.7  +MOVJ EC00284
SFTOF3D
SMOVL C00285 BC00285 V=666.7  +MOVJ EC00285
MOVJ C00286 BC00286 VJ=100.00  +MOVJ EC00286 VJ=100.00
MOVJ C00287 BC00287 VJ=100.00  +MOVJ EC00287 VJ=0.78
'
END
